{attribute addProperty BoxType "EK1122-0000-0018"}
{attribute addProperty Id "Beckhoff_EL4xxxsub_EK1100EK1100_179A0949162"}
{attribute addProperty CRC "3815418806"}
{attribute addProperty SizeInBites "16"}
{attribute addProperty SizeInBytes "2"}
TYPE Beckhoff_EL4xxxEK1122_E36AABB6 EXTENDS EK1122_179A0949 :
STRUCT
	{attribute addProperty Name "Beckhoff_EL4xxxsub_EK1100"}
	Beckhoff_EL4xxxsub_EK1100 : EK1100_179A0949;
END_STRUCT
END_TYPE

(* stored: Version 1.2.0.0, ProductVersion 3.1.4024.9
   DUT Beckhoff_EL4xxxEK1122_E36AABB6: Id {eccbf0b5-479d-4507-901f-c4b0a2483d48} *)
